TYPE
    ST_CSV : STRUCT
        Steps : ARRAY[1..MAX_STEP_COUNT] OF ST_CSV_Step;
    END_STRUCT
END_TYPE

(* stored: Version 1.1.0.1
   DUT ST_CSV: Id {39ac5a85-0924-465b-9add-bc2064d3e42c} *)
